# B&R Automation Studio project DevOpsDemo (part 2)

#### PackMLModuleStateManaging.cpp
```cpp
#include "PackMLModule.hpp"

		// -----------------------------------------------------------------------------

const char *internalInfoStateNames[] = { "Undefined",
	"Clearing",
	"Stopped",
	"Starting",
	"Idle",
	"Suspended",
	"Execute",
	"Stopping",
	"Aborting",
	"Aborted",
	"Holding",
	"Held",
	"Unholding",
	"Suspending",
	"Unsuspending",
	"Resetting",
	"Completing",
	"Completed",
	"",
	"",
	"",
	"",
	"",
	"",
	"",
	"",
	"",
	"",
	"",
	"",
	"Deactivating",
	"Deactivated",
	"Activating" };

const char *internalInfoModeNames[] = { "Undefined",
	"Production",
	"Maintenance",
	"Manual",
	""};

		// -----------------------------------------------------------------------------
		// we need to add complete cmd to the pattern
const unsigned long CMD_VALID_BIT_PATTERN_LIST[]
	= { 0,          0x00000080, 0x20004080, 0x000000C0, 0x000000C4, 0x0000A2C0,
	0x000092C0, 0x00000080, 0,          0x20000001, 0x000000C0, 0x000088C0,
	0x000000C0, 0x000000C0, 0x000000C0, 0x000000C0, 0x000000C0, 0x000040C0,
	0,          0,          0,          0,          0,          0,
	0,          0,          0,          0,          0,          0,
	0,          0x80000000, 0 };

// -----------------------------------------------------------------------------

PackMLModule* PackMLModule::getParentPtr(){
	if (!hasParent_)
		return nullptr;

	return pParentLink_;
}
// -----------------------------------------------------------------------------
PackMLModule* PackMLModule::getChildPtr(unsigned long int childIdx){
	if(childCount_ <= 0)
		return nullptr;

	return childLinks_[childIdx % childCount_];
}
// -----------------------------------------------------------------------------
PackMLModule* PackMLModule::getSiblingPtr(unsigned long int siblingIdx){
	if (!hasParent_)
		return nullptr;

	return pParentLink_->getChildPtr(siblingIdx);
}
// -----------------------------------------------------------------------------

PackMLModuleStateEnu PackMLModule::getChildCurrentState(unsigned long int childIndex){
	if(childCount_ <= 0)
		return ST_UNDEFINED;

	return childLinks_[childIndex % childCount_]->getCurrentState();
}
		// -----------------------------------------------------------------------------
long int PackMLModule::getChildCurrentSubState(unsigned long int childIndex){
	if(childCount_ <= 0)
		return 0;

	return childLinks_[childIndex % childCount_]->getCurrentSubState();
}
		// -----------------------------------------------------------------------------
bool PackMLModule::getChildStateComplete(unsigned long int childIndex){
	if(childCount_ <= 0)
		return false;

	return childLinks_[childIndex % childCount_]->getStateComplete();
}
		// -----------------------------------------------------------------------------
const char* PackMLModule::getChildName(unsigned long int childIndex){
	if(childCount_ <= 0)
		return "";

	return childLinks_[childIndex % childCount_]->getModuleName();
}
		// -----------------------------------------------------------------------------
PackMLModuleStateEnu PackMLModule::getSiblingCurrentState(unsigned long int siblingIndex){
	if (!hasParent_)
		return ST_UNDEFINED;

	return pParentLink_->getChildCurrentState(siblingIndex);
}
		// -----------------------------------------------------------------------------
long int PackMLModule::getSiblingCurrentSubState(unsigned long int siblingIndex){
	if (!hasParent_)
		return 0;

	return pParentLink_->getChildCurrentSubState(siblingIndex);
}
		// -----------------------------------------------------------------------------
bool PackMLModule::getSiblingStateComplete(unsigned long int siblingIndex){
	if (!hasParent_)
		return false;

	return pParentLink_->getChildStateComplete(siblingIndex);
}
		// -----------------------------------------------------------------------------
const char* PackMLModule::getSiblingName(unsigned long int siblingIndex){
	if (!hasParent_)
		return "";

	return pParentLink_->getChildName(siblingIndex);
}
		// -----------------------------------------------------------------------------
bool PackMLModule::isChild_(PackMLModule* pModule){
	for (unsigned short i = 0; i < childCount_; ++i) {
		if (childLinks_[i] == pModule) {
			return true;
		}
	}
	return false;
}
		// -----------------------------------------------------------------------------
unsigned long PackMLModule::getSiblingCount(){
	if (!hasParent_) {
		return 1;
	}
	return pParentLink_->getChildCount();
}
		// -----------------------------------------------------------------------------
bool PackMLModule::getSiblingsStateComplete(){
	if (!hasParent_) {
		return stateComplete_;
	}
	return pParentLink_->getChildrenStateComplete();
}

		// -----------------------------------------------------------------------------
bool PackMLModule::getChildrenStateComplete(){
	for (unsigned short i = 0; i < childCount_; ++i) {
		if (!childLinks_[i]->getStateComplete()) {
			return false;
		}
	}
	return true;
}
		// -----------------------------------------------------------------------------
PackMLModuleStateEnu PackMLModule::getParentCurrentState()
{
	if (!hasParent_) {
		return ST_UNDEFINED;
	}
	return pParentLink_->getCurrentState();
}

		// -----------------------------------------------------------------------------

long int PackMLModule::getParentCurrentSubState()
{
	if (!hasParent_) {
		return 0;
	}
	return pParentLink_->getCurrentSubState();
}

		// -----------------------------------------------------------------------------

const char *PackMLModule::getParentName()
{
	if (!hasParent_) {
		return "";
	}
	return pParentLink_->getModuleName();
}

bool PackMLModule::getParentStateComplete()
{
	if (!hasParent_) {
		return true;
	}
	return pParentLink_->getStateComplete();
}

		// -----------------------------------------------------------------------------

const char *PackMLModule::getCurrentStateStr() const
{
	return internalInfoStateNames[stateCurrent_];

}

const char *PackMLModule::getStateStr(PackMLModuleStateEnu state) const
{
	return internalInfoStateNames[state];
}

		// -----------------------------------------------------------------------------

		// -----------------------------------------------------------------------------

const char* PackMLModule::getCurrentModeName() const
{
	return internalInfoModeNames[modeCurrent_];
}

const char* PackMLModule::getModeName(signed long int modeId) const
{
	return internalInfoModeNames[modeId];
}

		// -----------------------------------------------------------------------------

// --------------------------------------------------------------------------

void PackMLModule::setNewModeCurrent(long int mode)
{
	modeCurrent_ = mode;

	for (unsigned short i = 0; i < childCount_; ++i) {
		childLinks_[i]->setNewModeCurrent(modeCurrent_);
	}
}

		// -----------------------------------------------------------------------------

bool PackMLModule::setCurrentMode(long int mode)
{

	// Check if the hierarchy is in synch
	if(!isModeChangePossible())
		return false;

	// update mode
	setNewModeCurrent(mode);
	// propagate mode to the children within one cycle
	return true;
}

		// -----------------------------------------------------------------------------

bool PackMLModule::isModeChangePossible()
{
	// What should the child do when it is not synchronized with the parent?
	if (!childrenInState_(stateCurrent_)) {
		return false;
	}

	for (unsigned short i = 0; i < childCount_; ++i) {
		if (!childLinks_[i]->isModeChangePossible()) {
			return false;
		}
	}

	return true;
}
		// -----------------------------------------------------------------------------

bool PackMLModule::childrenInState_(PackMLModuleStateEnu state)
{

	for (unsigned short i = 0; i < childCount_; ++i) {
		PackMLModuleStateEnu childState = childLinks_[i]->getCurrentState();
		if (childState != state && childState != ST_DEACTIVATED) {
			return false;
		}
	}
	return true;
}

		// -------------------------------------------------------------------------

bool PackMLModule::stateExistInPattern_(unsigned long stateBitPattern,
	PackMLModuleStateEnu state)
{
	if (state == ST_UNDEFINED) {
		return true;
	}
	unsigned long patternChecker = 1;
	return (stateBitPattern & (patternChecker << (state - 1)));
}

		// -------------------------------------------------------------------------

bool PackMLModule::cmdValid_(PackMLModuleStateEnu state)
{

	return stateExistInPattern_(CMD_VALID_BIT_PATTERN_LIST[stateCurrent_],
		state);
}

		// ------------------------------------------------------------------------

bool PackMLModule::isActingState(PackMLModuleStateEnu state)
{
	unsigned long actingStateBitPattern = 0xA000FAC5;

	return stateExistInPattern_(actingStateBitPattern, state);
}

		// -----------------------------------------------------------------------------

// from waiting state to acting state
void PackMLModule::executeCmd_(PackMLModuleStateEnu targetState)
{
	stateCurrent_ = targetState;
	// reset internal bools
	resetInternalCmds_();
	resetWaitingFor_();
	resetInterruptedBy_();
}

		// -----------------------------------------------------------------------------
// from acting state to waiting state
void PackMLModule::executeActingState_(PackMLModuleStateEnu targetState)
{
	if (childrenInSynch_(targetState)) {
		// Update the state
		stateCurrent_ = targetState;
		// reset internal bools
		resetInternalCmds_();
		resetWaitingFor_();
	}
}

		// -----------------------------------------------------------------------------
		// Checks if the children are in the desired state in case where they want to be
		// synchronized
bool PackMLModule::childrenInSynch_(PackMLModuleStateEnu targetState)
{

	for (unsigned long i = 0; i < childCount_; ++i) {
		if ((childLinks_[i]->getCurrentState() != targetState) && childLinks_[i]->needParentSynch(stateCurrent_)) {
			return false;
		}
	}
	return true;
}

		// -----------------------------------------------------------------------------

void PackMLModule::resetInternalCmds_()
{
	if(isActingState(stateCurrent_)){
		externalAbort_ = false;
		externalClear_ = false;
		externalStop_ = false;
		externalReset_ = false;
		externalStart_ = false;
		externalHold_ = false;
		externalUnhold_ = false;
		externalSuspend_ = false;
		externalUnsuspend_ = false;
		externalComplete_ = false;
		externalStateComplete_ = false;
	}

	activate_ = false;
	deactivate_ = false;

	abort_ = externalAbort_;
	clear_ = externalClear_;
	stop_ = externalStop_;
	reset_ = externalReset_;
	start_ = externalStart_;
	hold_ = externalHold_;
	unhold_ = externalUnhold_;
	suspend_ = externalSuspend_;
	unsuspend_ = externalUnsuspend_;
	complete_ = externalComplete_;
	stateComplete_ = false;

	oldAbort_ = false;
	oldClear_ = false;
	oldStop_ = false;
	oldReset_ = false;
	oldStart_ = false;
	oldHold_ = false;
	oldUnhold_ = false;
	oldSuspend_ = false;
	oldUnsuspend_ = false;
	oldComplete_ = false;
	oldStateComplete_ = false;

	timeInState_ = 0.0;
}

		// -----------------------------------------------------------------------------

void PackMLModule::escalateCmdAbort()
{
	if (escalateAbort_) {
		return pParentLink_->escalateCmdAbort();
	}
	abort_ = !overrideAbort_;
	externalAbort_ = abort_;
}
void PackMLModule::escalateCmdClear()
{
	if (escalateClear_) {
		return pParentLink_->escalateCmdClear();
	}
	clear_ = !overrideClear_;
	externalClear_ = clear_;
}
void PackMLModule::escalateCmdStop()
{
	if (escalateStop_) {
		return pParentLink_->escalateCmdStop();
	}
	stop_ = !overrideStop_;
	externalStop_ = stop_;
}
void PackMLModule::escalateCmdReset()
{
	if (escalateReset_) {
		return pParentLink_->escalateCmdReset();
	}
	reset_ = !overrideReset_;
	externalReset_ = reset_;
}
void PackMLModule::escalateCmdHold()
{
	if (escalateHold_) {
		return pParentLink_->escalateCmdHold();
	}
	hold_ = !overrideHold_;
	externalHold_ = hold_;
}
void PackMLModule::escalateCmdUnhold()
{
	if (escalateUnhold_) {
		return pParentLink_->escalateCmdUnhold();
	}
	unhold_ = !overrideUnhold_;
	externalUnhold_ = unhold_;
}
void PackMLModule::escalateCmdSuspend()
{
	if (escalateSuspend_) {
		return pParentLink_->escalateCmdSuspend();
	}
	suspend_ = !overrideSuspend_;
	externalSuspend_ = suspend_;
}
void PackMLModule::escalateCmdUnsuspend()
{
	if (escalateUnsuspend_) {
		return pParentLink_->escalateCmdUnsuspend();
	}
	unsuspend_ = !overrideUnsuspend_;
	externalUnsuspend_ = unsuspend_;
}
void PackMLModule::escalateCmdStart()
{
	if (escalateStart_) {
		return pParentLink_->escalateCmdStart();
	}
	start_ = !overrideStart_;
	externalStart_ = start_;
}
void PackMLModule::escalateCmdComplete()
{
	if (escalateComplete_) {
		return pParentLink_->escalateCmdComplete();
	}
	complete_ = !overrideComplete_;
	externalComplete_ = complete_;
}

// ----------------------------------------------------------------------------

void PackMLModule::propagateCmdAbort(bool root)
{
	abort_ = reactToAbort_ && !root;
	externalAbort_ = abort_;

	for (unsigned short i = 0; i < childCount_; ++i) {
		childLinks_[i]->propagateCmdAbort(false);
	}
}
void PackMLModule::propagateCmdClear(bool root)
{
	clear_ = reactToClear_ && !root;
	externalClear_ = clear_;

	for (unsigned short i = 0; i < childCount_; ++i) {
		childLinks_[i]->propagateCmdClear(false);
	}
}
void PackMLModule::propagateCmdStop(bool root)
{
	stop_ = reactToStop_ && !root;
	externalStop_ = stop_;

	for (unsigned short i = 0; i < childCount_; ++i) {
		childLinks_[i]->propagateCmdStop(false);
	}
}
void PackMLModule::propagateCmdReset(bool root)
{
	reset_ = reactToReset_ && !root;
	externalReset_ = reset_;

	for (unsigned short i = 0; i < childCount_; ++i) {
		childLinks_[i]->propagateCmdReset(false);
	}
}
void PackMLModule::propagateCmdHold(bool root)
{
	hold_ = reactToHold_ && !root;
	externalHold_ = hold_;

	for (unsigned short i = 0; i < childCount_; ++i) {
		childLinks_[i]->propagateCmdHold(false);
	}
}
void PackMLModule::propagateCmdUnhold(bool root)
{
	unhold_ = reactToUnhold_ && !root;
	externalUnhold_ = unhold_;

	for (unsigned short i = 0; i < childCount_; ++i) {
		childLinks_[i]->propagateCmdUnhold(false);
	}
}
void PackMLModule::propagateCmdSuspend(bool root)
{
	suspend_ = reactToSuspend_ && !root;
	externalSuspend_ = suspend_;

	for (unsigned short i = 0; i < childCount_; ++i) {
		childLinks_[i]->propagateCmdSuspend(false);
	}
}
void PackMLModule::propagateCmdUnsuspend(bool root)
{
	unsuspend_ = reactToUnsuspend_ && !root;
	externalUnsuspend_ = unsuspend_;

	for (unsigned short i = 0; i < childCount_; ++i) {
		childLinks_[i]->propagateCmdUnsuspend(false);
	}
}
void PackMLModule::propagateCmdStart(bool root)
{
	start_ = reactToStart_ && !root;
	externalStart_ = start_;

	for (unsigned short i = 0; i < childCount_; ++i) {
		childLinks_[i]->propagateCmdStart(false);
	}
}
void PackMLModule::propagateCmdComplete(bool root)
{
	complete_ = reactToComplete_ && !root;
	externalComplete_ = complete_;

	for (unsigned short i = 0; i < childCount_; ++i) {
		childLinks_[i]->propagateCmdComplete(false);
	}
}

// ----------------------------------------------------------------------------

bool PackMLModule::evaluateCmdAbort(bool& newCmd)
{
	if (newCmd && !oldAbort_) {
		oldAbort_ = true;
		return setCmd_(ST_ABORTING);
	}
	else if (!newCmd && oldAbort_) {
		oldAbort_ = false;
		resetCmd_(ST_ABORTING);
	}
	return true;
}
bool PackMLModule::evaluateCmdStop(bool& newCmd)
{
	if (newCmd && !oldStop_) {
		oldStop_ = true;
		return setCmd_(ST_STOPPING);
	}
	else if (!newCmd && oldStop_) {
		oldStop_ = false;
		resetCmd_(ST_STOPPING);
	}
	return true;
}
bool PackMLModule::evaluateCmdClear(bool& newCmd)
{
	if (newCmd && !oldClear_) {
		oldClear_ = true;
		return setCmd_(ST_CLEARING);
	}
	else if (!newCmd && oldClear_) {
		oldClear_ = false;
		resetCmd_(ST_CLEARING);
	}
	return true;
}
bool PackMLModule::evaluateCmdReset(bool& newCmd)
{
	if (newCmd && !oldReset_) {
		oldReset_ = true;
		return setCmd_(ST_RESETTING);
	}
	else if (!newCmd && oldReset_) {
		oldReset_ = false;
		resetCmd_(ST_RESETTING);
	}
	return true;
}
bool PackMLModule::evaluateCmdStart(bool& newCmd)
{
	if (newCmd && !oldStart_) {
		oldStart_ = true;
		return setCmd_(ST_STARTING);
	}
	else if (!newCmd && oldStart_) {
		oldStart_ = false;
		resetCmd_(ST_STARTING);
	}
	return true;
}
bool PackMLModule::evaluateCmdSuspend(bool& newCmd)
{
	if (newCmd && !oldSuspend_) {
		oldSuspend_ = true;
		return setCmd_(ST_SUSPENDING);
	}
	else if (!newCmd && oldSuspend_) {
		oldSuspend_ = false;
		resetCmd_(ST_SUSPENDING);
	}
	return true;
}
bool PackMLModule::evaluateCmdUnsuspend(bool& newCmd)
{
	if (newCmd && !oldUnsuspend_) {
		oldUnsuspend_ = true;
		return setCmd_(ST_UNSUSPENDING);
	}
	else if (!newCmd && oldUnsuspend_) {
		oldUnsuspend_ = false;
		resetCmd_(ST_UNSUSPENDING);
	}
	return true;
}
bool PackMLModule::evaluateCmdHold(bool& newCmd)
{
	if (newCmd && !oldHold_) {
		oldHold_ = true;
		return setCmd_(ST_HOLDING);
	}
	else if (!newCmd && oldHold_) {
		oldHold_ = false;
		resetCmd_(ST_HOLDING);
	}
	return true;
}
bool PackMLModule::evaluateCmdUnhold(bool& newCmd)
{
	if (newCmd && !oldUnhold_) {
		oldUnhold_ = true;
		return setCmd_(ST_UNHOLDING);
	}
	else if (!newCmd && oldUnhold_) {
		oldUnhold_ = false;
		resetCmd_(ST_UNHOLDING);
	}
	return true;
}
bool PackMLModule::evaluateCmdComplete(bool& newCmd)
{
	if (newCmd && !oldComplete_) {
		oldComplete_ = true;
		return setCmd_(ST_COMPLETING);
	}
	else if (!newCmd && oldComplete_) {
		oldComplete_ = false;
		resetCmd_(ST_COMPLETING);
	}
	return true;
}
bool PackMLModule::evaluateCmdStateComplete(bool& newCmd)
{
	if (newCmd && !oldStateComplete_) {
		oldStateComplete_ = true;
		return setCmd_(ST_UNDEFINED);
	}
	else if (!newCmd && oldStateComplete_) {
		oldStateComplete_ = false;
		resetCmd_(ST_UNDEFINED);
	}
	return true;
}

bool PackMLModule::setCmdAbort(){
	return setCmd_(ST_ABORTING);
}
bool PackMLModule::setCmdStop(){
	return setCmd_(ST_STOPPING);
}
bool PackMLModule::setCmdClear(){
	return setCmd_(ST_CLEARING);
}
bool PackMLModule::setCmdReset(){
	return setCmd_(ST_RESETTING);
}
bool PackMLModule::setCmdStart(){
	return setCmd_(ST_STARTING);
}
bool PackMLModule::setCmdSuspend(){
	return setCmd_(ST_SUSPENDING);
}
bool PackMLModule::setCmdUnsuspend(){
	return setCmd_(ST_UNSUSPENDING);
}
bool PackMLModule::setCmdHold(){
	return setCmd_(ST_HOLDING);
}
bool PackMLModule::setCmdUnhold(){
	return setCmd_(ST_UNHOLDING);
}
bool PackMLModule::setCmdComplete(){
	return setCmd_(ST_COMPLETING);
}
bool PackMLModule::setCmdStateComplete(){
	return setCmd_(ST_UNDEFINED);
}

void PackMLModule::resetCmdAbort(){
	return resetCmd_(ST_ABORTING);
}
void PackMLModule::resetCmdStop(){
	return resetCmd_(ST_STOPPING);
}
void PackMLModule::resetCmdClear(){
	return resetCmd_(ST_CLEARING);
}
void PackMLModule::resetCmdReset(){
	return resetCmd_(ST_RESETTING);
}
void PackMLModule::resetCmdStart(){
	return resetCmd_(ST_STARTING);
}
void PackMLModule::resetCmdSuspend(){
	return resetCmd_(ST_SUSPENDING);
}
void PackMLModule::resetCmdUnsuspend(){
	return resetCmd_(ST_UNSUSPENDING);
}
void PackMLModule::resetCmdHold(){
	return resetCmd_(ST_HOLDING);
}
void PackMLModule::resetCmdUnhold(){
	return resetCmd_(ST_UNHOLDING);
}
void PackMLModule::resetCmdComplete(){
	return resetCmd_(ST_COMPLETING);
}
void PackMLModule::resetCmdStateComplete(){
	return resetCmd_(ST_UNDEFINED);
}

		// -----------------------------------------------------------------------------

bool PackMLModule::setCmd_(PackMLModuleStateEnu targetActingState) // NOLINT
{

	bool cmdValid = cmdValid_(targetActingState);

	switch (targetActingState) { // NOCCM
		case ST_CLEARING:
			if (overrideClear_ && !escalateClear_) {
				return false; // error code
			}
			if (hasParent_ && escalateClear_ && cmdValid) {
				pParentLink_->escalateCmdClear();
				setInterruptedBy_(ST_CLEARING);
			}
			clear_ = !overrideClear_; //!overrideAbort_ || !escalateAbort_;
			break;

		case ST_STARTING:
			if (overrideStart_ && !escalateStart_) {
				return false; // error code
			}
			if (hasParent_ && escalateStart_ && cmdValid) {
				pParentLink_->escalateCmdStart();
				setInterruptedBy_(ST_STARTING);
			}
			start_ = !overrideStart_;
			break;

		case ST_STOPPING:
			if (overrideStop_ && !escalateStop_) {
				return false; // error code
			}
			if (hasParent_ && escalateStop_) {
				pParentLink_->escalateCmdStop();
			}
			if(cmdValid){
				setInterruptedBy_(ST_STOPPING);
				stop_ = !overrideStop_;
			}
			break;

		case ST_ABORTING:
			if (overrideAbort_ && !escalateAbort_) {
				return false; // error code
			}
			if (hasParent_ && escalateAbort_) {
				pParentLink_->escalateCmdAbort();
			}

			if(cmdValid){
				setInterruptedBy_(ST_ABORTING);
				abort_ = !overrideAbort_;
			}
			break;

		case ST_HOLDING:
			if (overrideHold_ && !escalateHold_) {
				return false; // error code
			}
			if (hasParent_ && escalateHold_) {
				pParentLink_->escalateCmdHold();
			}
			if(cmdValid){
				setInterruptedBy_(ST_HOLDING);
				hold_ = !overrideHold_;
			}
			break;

		case ST_UNHOLDING:
			if (overrideUnhold_ && !escalateUnhold_) {
				return false; // error code
			}
			if (hasParent_ && escalateUnhold_ && cmdValid) {
				pParentLink_->escalateCmdUnhold();
				setInterruptedBy_(ST_UNHOLDING);
			}
			unhold_ = !overrideUnhold_;
			break;

		case ST_SUSPENDING:
			if (overrideSuspend_ && !escalateSuspend_) {
				return false; // error code
			}
			if (hasParent_ && escalateSuspend_) {
				pParentLink_->escalateCmdSuspend();
			}
			if(cmdValid){
				setInterruptedBy_(ST_SUSPENDING);
				suspend_ = !overrideSuspend_;
			}
			break;

		case ST_UNSUSPENDING:
			if (overrideUnsuspend_ && !escalateUnsuspend_) {
				return false; // error code
			}
			if (hasParent_ && escalateUnsuspend_ && cmdValid) {
				pParentLink_->escalateCmdUnsuspend();
				setInterruptedBy_(ST_UNSUSPENDING);
			}
			unsuspend_ = !overrideUnsuspend_;
			break;

		case ST_RESETTING:
			if (overrideReset_ && !escalateReset_) {
				return false; // error code
			}
			if (hasParent_ && escalateReset_ && cmdValid) {
				pParentLink_->escalateCmdReset();
				setInterruptedBy_(ST_RESETTING);
			}
			reset_ = !overrideReset_;
			break;

		case ST_COMPLETING:
			// check if the state group is configured
			if (overrideComplete_ && !escalateComplete_) {
				return false; // error code
			}
			if (hasParent_ && escalateComplete_) {
				pParentLink_->escalateCmdComplete();
			}
			if(cmdValid){
				setInterruptedBy_(ST_COMPLETING);
				complete_ = !overrideComplete_;
			}
			break;

		case ST_UNDEFINED:
			stateComplete_ = true;
			break;

		default:
			break;
	}

	return true;
}

		// -----------------------------------------------------------------------------

void PackMLModule::resetCmd_(PackMLModuleStateEnu targetActingState)
{

	switch (targetActingState) { // NOCCM
		case ST_CLEARING:
			clear_ = externalClear_;
			break;

		case ST_STARTING:
			start_ = externalStart_;
			break;

		case ST_STOPPING:
			stop_ = externalStop_;
			break;

		case ST_ABORTING:
			abort_ = externalAbort_;
			break;

		case ST_HOLDING:
			hold_ = externalHold_;
			break;

		case ST_UNHOLDING:
			unhold_ = externalUnhold_;
			break;

		case ST_SUSPENDING:
			suspend_ = externalSuspend_;
			break;

		case ST_UNSUSPENDING:
			unsuspend_ = externalUnsuspend_;
			break;

		case ST_RESETTING:
			reset_ = externalReset_;
			break;

		case ST_COMPLETING:
			complete_ = externalComplete_;
			break;

		case ST_UNDEFINED:
			stateComplete_ = externalStateComplete_;
			break;

		default:
			break;
	}
}

		// -----------------------------------------------------------------------------

		// if parent synchronization needed
bool PackMLModule::needParentSynch(PackMLModuleStateEnu state)
{
	if (hierarchyLevel_ == 0) {
		return true;
	}

	switch (stateCurrent_) { // NOCCM

		case ST_CLEARING:
			switch (state) { // NOCCM
				case ST_ABORTING:
					return overrideAbort_ || reactToAbort_;
				case ST_CLEARING:
					return overrideClear_ || reactToClear_;
				default:
					break;
			}
			break;

		case ST_STOPPED:
			switch (state) { // NOCCM
				case ST_ABORTING:
					return overrideAbort_ || reactToAbort_;
				case ST_RESETTING:
					return overrideReset_ || reactToReset_;
				default:
					break;
			}
			break;

		case ST_IDLE:
			switch (state) { // NOCCM
				case ST_ABORTING:
					return overrideAbort_ || reactToAbort_;
				case ST_STOPPING:
					return overrideStop_ || reactToStop_;
				case ST_STARTING:
					return overrideStart_ || reactToStart_;
				default:
					break;
			}
			break;

		case ST_SUSPENDED:
			switch (state) { // NOCCM
				case ST_ABORTING:
					return overrideAbort_ || reactToAbort_;
				case ST_STOPPING:
					return overrideStop_ || reactToStop_;
				case ST_UNSUSPENDING:
					return overrideUnsuspend_ || reactToUnsuspend_;
				case ST_HOLDING:
					return overrideHold_ || reactToHold_;
				case ST_COMPLETING:
					return overrideComplete_ || reactToComplete_;
				default:
					break;
			}
			break;

		case ST_EXECUTE:
			switch (state) { // NOCCM
				case ST_ABORTING:
					return overrideAbort_ || reactToAbort_;
				case ST_STOPPING:
					return overrideStop_ || reactToStop_;
				case ST_SUSPENDING:
					return overrideSuspend_ || reactToSuspend_;
				case ST_HOLDING:
					return overrideHold_ || reactToHold_;
				case ST_COMPLETING:
					return overrideComplete_ || reactToComplete_;
				default:
					break;
			}
			break;

		case ST_STOPPING:
			switch (state) { // NOCCM
				case ST_ABORTING:
					return overrideAbort_ || reactToAbort_;
				case ST_STOPPING:
					return overrideStop_ || reactToStop_;
				default:
					break;
			}
			break;

		case ST_ABORTING:
			switch (state) { // NOCCM
				case ST_ABORTING:
					return overrideAbort_ || reactToAbort_;
				default:
					break;
			}
			break;

		case ST_ABORTED:
			switch (state) { // NOCCM
				case ST_CLEARING:
					return overrideClear_ || reactToClear_;
				default:
					break;
			}
			break;

		case ST_HELD:
			switch (state) { // NOCCM
				case ST_ABORTING:
					return overrideAbort_ || reactToAbort_;
				case ST_STOPPING:
					return overrideStop_ || reactToStop_;
				case ST_UNHOLDING:
					return overrideUnhold_ || reactToUnhold_;
				case ST_COMPLETING:
					return overrideComplete_ || reactToComplete_;
				default:
					break;
			}
			break;

		case ST_SUSPENDING:
			switch (state) { // NOCCM
				case ST_ABORTING:
					return overrideAbort_ || reactToAbort_;
				case ST_STOPPING:
					return overrideStop_ || reactToStop_;
				case ST_SUSPENDING:
					return overrideSuspend_ || reactToSuspend_;
				default:
					break;
			}
			break;
		case ST_UNSUSPENDING:
			switch (state) { // NOCCM
				case ST_ABORTING:
					return overrideAbort_ || reactToAbort_;
				case ST_STOPPING:
					return overrideStop_ || reactToStop_;
				case ST_UNSUSPENDING:
					return overrideUnsuspend_ || reactToUnsuspend_;
				default:
					break;
			}
			break;
		case ST_COMPLETING:
			switch (state) { // NOCCM
				case ST_ABORTING:
					return overrideAbort_ || reactToAbort_;
				case ST_STOPPING:
					return overrideStop_ || reactToStop_;
				case ST_COMPLETING:
					return overrideComplete_ || reactToComplete_;
				default:
					break;
			}
			break;
		case ST_STARTING:
			switch (state) { // NOCCM
				case ST_ABORTING:
					return overrideAbort_ || reactToAbort_;
				case ST_STOPPING:
					return overrideStop_ || reactToStop_;
				case ST_STARTING:
					return overrideStart_ || reactToStart_;
				default:
					break;
			}
			break;
		case ST_HOLDING:
			switch (state) { // NOCCM
				case ST_ABORTING:
					return overrideAbort_ || reactToAbort_;
				case ST_STOPPING:
					return overrideStop_ || reactToStop_;
				case ST_HOLDING:
					return overrideHold_ || reactToHold_;
				default:
					break;
			}
			break;
		case ST_UNHOLDING:
			switch (state) { // NOCCM
				case ST_ABORTING:
					return overrideAbort_ || reactToAbort_;
				case ST_STOPPING:
					return overrideStop_ || reactToStop_;
				case ST_UNHOLDING:
					return overrideUnhold_ || reactToUnhold_;
				default:
					break;
			}
			break;

		case ST_RESETTING:
			switch (state) { // NOCCM
				case ST_ABORTING:
					return overrideAbort_ || reactToAbort_;
				case ST_STOPPING:
					return overrideStop_ || reactToStop_;
				case ST_RESETTING:
					return overrideReset_ || reactToReset_;
				default:
					break;
			}
			break;

		case ST_COMPLETE:
			switch (state) { // NOCCM
				case ST_ABORTING:
					return overrideAbort_ || reactToAbort_;
				case ST_STOPPING:
					return overrideStop_ || reactToStop_;
				case ST_RESETTING:
					return overrideReset_ || reactToReset_;
				default:
					break;
			}
			break;

		default:
			break;
	}

	return false;
}

// -----------------------------------------------------------------------------
// decide if reacto to only should when parent + 1 state in front of child. e.g. instead of ST_ABORTING and ST_ABORTED --> only ST_ABORTING
void PackMLModule::checkParentStateCondition_()
{
	if (hierarchyLevel_ == 0) {
		return;
	}

	PackMLModuleStateEnu parentState = getParentCurrentState();

	if (parentState == stateCurrent_) {
		return;
	}

	switch (stateCurrent_) { // NOCCM
		case ST_CLEARING:
			switch (parentState) { // NOCCM
				case ST_ABORTING:
					abort_ = overrideAbort_ || abort_ || reactToAbort_;
					break;
				case ST_ABORTED:
					abort_ = overrideAbort_ || abort_;
					break;
				default:
					break;
			}
			break;

		case ST_STOPPED:
			switch (parentState) { // NOCCM
				case ST_ABORTING:
					abort_ = overrideAbort_ || abort_ || reactToAbort_;
					break;
				case ST_ABORTED:
					abort_ = overrideAbort_ || abort_;
					break;

				case ST_DEACTIVATING:
				case ST_DEACTIVATED:
					deactivate_ = (activationCondition_ == 1);
					break;

				case ST_RESETTING:
					reset_ = overrideReset_ || reset_ || reactToReset_;
					break;

				case ST_IDLE:
				case ST_STARTING:
				case ST_SUSPENDED:
				case ST_EXECUTE:
				case ST_HOLDING:
				case ST_HELD:
				case ST_UNHOLDING:
				case ST_SUSPENDING:
				case ST_UNSUSPENDING:
				case ST_COMPLETING:
				case ST_COMPLETE:
					reset_ = overrideReset_ || reset_;
					break;

				default:
					break;
			}
			break;

		case ST_IDLE:
			switch (parentState) { // NOCCM
				case ST_ABORTING:
					abort_ = overrideAbort_ || abort_ || reactToAbort_;
					break;
				case ST_ABORTED:
					abort_ = overrideAbort_ || abort_;
					break;

				case ST_CLEARING:
					stop_ = overrideStop_ || stop_;
					abort_ = (overrideAbort_ || abort_) && !stop_;
					break;

				case ST_STOPPING:
					stop_ = overrideStop_ || stop_ || reactToStop_;
					break;
				case ST_STOPPED:
					stop_ = overrideStop_ || stop_;
					break;

				case ST_DEACTIVATING:
				case ST_DEACTIVATED:
				case ST_ACTIVATING:
					stop_ = overrideStop_ || stop_;
					abort_ = (overrideAbort_ || abort_) && !stop_;
					break;

				case ST_STARTING:
					start_ = overrideStart_ || start_ || reactToStart_;
					break;

				case ST_EXECUTE:
				case ST_SUSPENDED:
				case ST_HOLDING:
				case ST_HELD:
				case ST_UNHOLDING:
				case ST_SUSPENDING:
				case ST_UNSUSPENDING:
				case ST_COMPLETING:
				case ST_COMPLETE:
					start_ = overrideStart_ || start_;
					break;

				default:
					break;
			}
			break;

		case ST_SUSPENDED:
			switch (parentState) { // NOCCM
				case ST_ABORTING:
					abort_ = overrideAbort_ || abort_ || reactToAbort_;
					break;
				case ST_ABORTED:
					abort_ = overrideAbort_ || abort_;
					break;

				case ST_CLEARING:
					stop_ = overrideStop_ || stop_;
					abort_ = (overrideAbort_ || abort_) && !stop_;
					break;

				case ST_STOPPING:
					stop_ = overrideStop_ || stop_ || reactToStop_;
					break;
				case ST_STOPPED:
					stop_ = overrideStop_ || stop_;
					break;

				case ST_UNSUSPENDING:
					unsuspend_ = overrideUnsuspend_ || unsuspend_ || reactToUnsuspend_;
					break;

				case ST_DEACTIVATING:
				case ST_DEACTIVATED:
				case ST_ACTIVATING:
					stop_ = overrideStop_ || stop_;
					abort_ = (overrideAbort_ || abort_) && !stop_;
					break;

				case ST_RESETTING:
				case ST_IDLE: // **********************
					unsuspend_ = overrideUnsuspend_ || unsuspend_;
					stop_ = (overrideStop_ || stop_) && !unsuspend_;
					break;

				case ST_COMPLETING:
					complete_ = overrideComplete_ || complete_ || reactToComplete_;
					break;
				case ST_COMPLETE:
					complete_ = overrideComplete_ || complete_;
					break;

				case ST_HOLDING:
					hold_ = overrideHold_ || hold_ || reactToHold_;
					break;
				case ST_HELD:
					hold_ = overrideHold_ || hold_;
					break;

				case ST_EXECUTE:
				case ST_STARTING:
				case ST_UNHOLDING:
					unsuspend_ = overrideUnsuspend_ || unsuspend_;
					break;

				default:
					break;
			}
			break;

		case ST_EXECUTE:
			switch (parentState) { // NOCCM
				case ST_ABORTING:
					abort_ = overrideAbort_ || abort_ || reactToAbort_;
					break;
				case ST_ABORTED:
					abort_ = overrideAbort_ || abort_;
					break;

				case ST_CLEARING:
					stop_ = overrideStop_ || stop_;
					abort_ = (overrideAbort_ || abort_) && !stop_;
					break;

				case ST_STOPPING:
					stop_ = overrideStop_ || stop_ || reactToStop_;
					break;

				case ST_STOPPED:
					stop_ = overrideStop_ || stop_;
					break;

				case ST_SUSPENDING:
					suspend_ = overrideSuspend_ || suspend_ || reactToSuspend_;
					break;

				case ST_SUSPENDED:
					suspend_ = overrideSuspend_ || suspend_;
					break;

				case ST_HOLDING:
					hold_ = overrideHold_ || hold_ || reactToHold_;
					break;

				case ST_HELD:
					hold_ = overrideHold_ || hold_;
					break;

				case ST_COMPLETING:
					complete_ = overrideComplete_ || complete_ || reactToComplete_;
					break;

				case ST_COMPLETE:
					complete_ = overrideComplete_ || complete_;
					break;

				case ST_DEACTIVATING:
				case ST_DEACTIVATED:
				case ST_ACTIVATING:
					stop_ = overrideStop_ || stop_;
					abort_ = (overrideAbort_ || abort_) && !stop_;
					break;

				case ST_RESETTING:
				case ST_IDLE:
					complete_ = overrideComplete_ || complete_;
					stop_ = (overrideStop_ || stop_) && !complete_;
					break;

				default:
					break;
			}
			break;

		case ST_STOPPING:
			switch (parentState) { // NOCCM
				case ST_ABORTING:
					abort_ = overrideAbort_ || abort_ || reactToAbort_;
					break;
				case ST_ABORTED:
					abort_ = overrideAbort_ || abort_;
					break;
				default:
					break;
			}
			break;

		case ST_ABORTED:
			switch (parentState) { // NOCCM
				case ST_DEACTIVATING:
				case ST_DEACTIVATED:
					deactivate_ = (activationCondition_ == 1);
					break;

				case ST_CLEARING:
					clear_ = overrideClear_ || clear_ || reactToClear_;
					break;

				case ST_STOPPED:
				case ST_STARTING:
				case ST_IDLE:
				case ST_SUSPENDED:
				case ST_EXECUTE:
				case ST_STOPPING:
				case ST_HOLDING:
				case ST_HELD:
				case ST_UNHOLDING:
				case ST_SUSPENDING:
				case ST_UNSUSPENDING:
				case ST_RESETTING:
				case ST_COMPLETING:
				case ST_COMPLETE:
				case ST_ACTIVATING:
					clear_ = overrideClear_ || clear_;
					break;

				default:
					break;
			}
			break;

		case ST_HELD:
			switch (parentState) { // NOCCM
				case ST_ABORTING:
					abort_ = overrideAbort_ || abort_ || reactToAbort_;
					break;
				case ST_ABORTED:
					abort_ = overrideAbort_ || abort_;
					break;

				case ST_CLEARING:
					stop_ = overrideStop_ || stop_;
					abort_ = (overrideAbort_ || abort_) && !stop_;
					break;

				case ST_STOPPING:
					stop_ = overrideStop_ || stop_ || reactToStop_;
					break;

				case ST_STOPPED:
					stop_ = overrideStop_ || stop_;
					break;

				case ST_UNHOLDING:
					unhold_ = overrideUnhold_ || unhold_ || reactToUnhold_;
					break;

				case ST_DEACTIVATING:
				case ST_DEACTIVATED:
				case ST_ACTIVATING:
					stop_ = overrideStop_ || stop_;
					abort_ = (overrideAbort_ || abort_) && !stop_;
					break;

				case ST_RESETTING:
				case ST_IDLE: // **********************
					unhold_ = overrideUnhold_ || unhold_;
					stop_ = (overrideStop_ || stop_) && !unhold_;
					break;

				case ST_COMPLETING:
					complete_ = overrideComplete_ || complete_ || reactToComplete_;
					break;
				case ST_COMPLETE:
					complete_ = overrideComplete_ || complete_;
					break;

				case ST_EXECUTE:
				case ST_SUSPENDING:
				case ST_SUSPENDED:
				case ST_UNSUSPENDING:
				case ST_STARTING:
					unhold_ = overrideUnhold_ || unhold_;
					break;

				default:
					break;
			}
			break;

		case ST_STARTING:
		case ST_HOLDING:
		case ST_UNHOLDING:
		case ST_SUSPENDING:
		case ST_UNSUSPENDING:
			switch (parentState) { // NOCCM
				case ST_ABORTING:
					abort_ = overrideAbort_ || abort_ || reactToAbort_;
					break;

				case ST_ABORTED:
					abort_ = overrideAbort_ || abort_;
					break;

				case ST_CLEARING:
					stop_ = overrideStop_ || stop_;
					abort_ = (overrideAbort_ || abort_) && !stop_;
					break;

				case ST_STOPPING:
					stop_ = overrideStop_ || stop_ || reactToStop_;
					break;

				case ST_STOPPED:
					stop_ = overrideStop_ || stop_;
					break;

				case ST_DEACTIVATING:
				case ST_DEACTIVATED:
				case ST_ACTIVATING:
					stop_ = overrideStop_ || stop_;
					abort_ = (overrideAbort_ || abort_) && !stop_;
					break;

				case ST_RESETTING:
				case ST_IDLE:
					stop_ = overrideStop_ || stop_;
					break;

				default:
					break;
			}
			break;

		case ST_RESETTING:
		case ST_COMPLETING:
			switch (parentState) { // NOCCM
				case ST_ABORTING:
					abort_ = overrideAbort_ || abort_ || reactToAbort_;
					break;
				case ST_ABORTED:
					abort_ = overrideAbort_ || abort_;
					break;

				case ST_CLEARING:
					stop_ = overrideStop_ || stop_;
					abort_ = (overrideAbort_ || abort_) && !stop_;
					break;

				case ST_STOPPING:
					stop_ = overrideStop_ || stop_ || reactToStop_;
					break;

				case ST_STOPPED:
					stop_ = overrideStop_ || stop_;
					break;

				case ST_DEACTIVATING:
				case ST_DEACTIVATED:
				case ST_ACTIVATING:
					stop_ = overrideStop_ || stop_;
					abort_ = (overrideAbort_ || abort_) && !stop_;
					break;

				default:
					break;
			}
			break;

		case ST_COMPLETE:
			switch (parentState) { // NOCCM
				case ST_ABORTING:
					abort_ = overrideAbort_ || abort_ || reactToAbort_;
					break;
				case ST_ABORTED:
					abort_ = overrideAbort_ || abort_;
					break;

				case ST_CLEARING:
					stop_ = overrideStop_ || stop_;
					abort_ = (overrideAbort_ || abort_) && !stop_;
					break;

				case ST_STOPPING:
					stop_ = overrideStop_ || stop_ || reactToStop_;
					break;

				case ST_STOPPED:
					stop_ = overrideStop_ || stop_;
					break;

				case ST_DEACTIVATING:
				case ST_DEACTIVATED:
				case ST_ACTIVATING:
					stop_ = overrideStop_ || stop_;
					abort_ = (overrideAbort_ || abort_) && !stop_;
					break;

				case ST_RESETTING:
					reset_ = overrideReset_ || reset_ || reactToReset_;
					break;

				case ST_IDLE:
				case ST_STARTING:
				case ST_SUSPENDED:
				case ST_EXECUTE:
				case ST_HOLDING:
				case ST_HELD:
				case ST_UNHOLDING:
				case ST_SUSPENDING:
				case ST_UNSUSPENDING:
					reset_ = overrideReset_ || reset_;
					break;

				default:
					break;
			}
			break;

		case ST_DEACTIVATED:
			if (parentState != ST_DEACTIVATING) {
				activate_ = (activationCondition_ == 1);
			}
			break;

		default:
			break;
	}

}

void PackMLModule::resetWaitingFor_()
{
	if((waitingForIndex_ == moduleIndex_) && hasParent_){
		pParentLink_->escalateResetWaitingFor(moduleIndex_);
	}

	waitingForIndex_ = 0xFFFFFFFF;
	waitingForLevel_ = 0;
}

void PackMLModule::escalateResetWaitingFor(unsigned long int waitingForIndex){

	if(waitingForIndex == waitingForIndex_){
		waitingForIndex_ = 0xFFFFFFFF;
		waitingForLevel_ = 0;
	}

	if(hasParent_){
		pParentLink_->escalateResetWaitingFor(waitingForIndex);
	}

}

void PackMLModule::setWaitingFor_(PackMLModuleStateEnu cmdState)
{
	// escallate
	if(hierarchyLevel_ >= waitingForLevel_){
		waitingForIndex_ = moduleIndex_;
		waitingForLevel_ = hierarchyLevel_;

		if(hasParent_ && needParentSynch(cmdState)){
			pParentLink_->escalateWaitingFor(waitingForIndex_, waitingForLevel_, cmdState);
		}
	}
}

void PackMLModule::escalateWaitingFor(unsigned long int waitingForIndex, unsigned short int waitingForLevel, PackMLModuleStateEnu cmdState){

	if(waitingForLevel >= waitingForLevel_){
		waitingForIndex_ = waitingForIndex;
		waitingForLevel_ = waitingForLevel;

		if(hasParent_ && needParentSynch(cmdState)){
			pParentLink_->escalateWaitingFor(waitingForIndex_, waitingForLevel_, cmdState);
		}
	}
}

//void PackMLModule::escalateWaitingFor(unsigned long int moduleIndex)
//{
//	if (escalateStart_) {
//		return pParentLink_->escalateCmdStart();
//	}
//}

	//	 -----------------------------------------------------------------------------

void PackMLModule::resetInterruptedBy_()
{
	switch(interruptedInState_){
		case ST_EXECUTE:
			if(stateCurrent_ == ST_ABORTING || stateCurrent_ == ST_SUSPENDING || stateCurrent_ == ST_HOLDING || stateCurrent_ == ST_STOPPING || stateCurrent_ == ST_COMPLETING)
				return;
			break;

		case ST_STOPPED:
			if(stateCurrent_ == ST_ABORTING || stateCurrent_ == ST_RESETTING)
				return;
			break;

		case ST_IDLE:
			if(stateCurrent_ == ST_ABORTING || stateCurrent_ == ST_STOPPING || stateCurrent_ == ST_STARTING)
				return;
			break;

		case ST_HELD:
			if(stateCurrent_ == ST_ABORTING || stateCurrent_ == ST_STOPPING || stateCurrent_ == ST_UNHOLDING)
				return;
			break;

		case ST_SUSPENDED:
			if(stateCurrent_ == ST_ABORTING || stateCurrent_ == ST_STOPPING || stateCurrent_ == ST_UNSUSPENDING)
				return;
			break;

		case ST_ABORTED:
			if(stateCurrent_ == ST_CLEARING)
				return;
			break;

		case ST_COMPLETE:
			if(stateCurrent_ == ST_ABORTING || stateCurrent_ == ST_STOPPING || stateCurrent_ == ST_RESETTING)
				return;
			break;

	//	case ST_RESETTING: ST_STARTING: ST_HOLDING: ST_UNHOLDING: ST_SUSPENDING: ST_UNSUSPENDING: ST_COMPLETING: ST_STOPPING: ST_ABORTING: ST_CLEARING:
		default:
			if(stateCurrent_ == ST_ABORTING || stateCurrent_ == ST_STOPPING)
				return;
			break;
	}

	interruptedByIndex_ = 0xFFFFFFFF;
	interruptedInState_ = ST_UNDEFINED;
	interruptedInSubState_ = 0;
}

void PackMLModule::setInterruptedBy_(PackMLModuleStateEnu cmdState)
{
	escalateInterruptedBy(moduleIndex_, stateCurrent_, subStateCurrent_, cmdState);
}

void PackMLModule::escalateInterruptedBy(unsigned long int moduleIndex, PackMLModuleStateEnu state, signed long int subState, PackMLModuleStateEnu cmdState)
{
	switch (cmdState) { // NOCCM
		case ST_CLEARING:
			if (hasParent_ && escalateClear_) {
				return pParentLink_->escalateInterruptedBy(moduleIndex, state, subState, cmdState);
			}
			break;

		case ST_STARTING:
			if (hasParent_ && escalateStart_) {
				return pParentLink_->escalateInterruptedBy(moduleIndex, state, subState, cmdState);
			}
			break;

		case ST_STOPPING:
			if (hasParent_ && escalateStop_) {
				return pParentLink_->escalateInterruptedBy(moduleIndex, state, subState, cmdState);
			}
			break;

		case ST_ABORTING:
			if (hasParent_ && escalateAbort_) {
				return pParentLink_->escalateInterruptedBy(moduleIndex, state, subState, cmdState);
			}
			break;

		case ST_HOLDING:
			if (hasParent_ && escalateHold_) {
				return pParentLink_->escalateInterruptedBy(moduleIndex, state, subState, cmdState);
			}
			break;

		case ST_UNHOLDING:
			if (hasParent_ && escalateUnhold_) {
				return pParentLink_->escalateInterruptedBy(moduleIndex, state, subState, cmdState);
			}
			break;

		case ST_SUSPENDING:
			if (hasParent_ && escalateSuspend_) {
				return pParentLink_->escalateInterruptedBy(moduleIndex, state, subState, cmdState);
			}
			break;

		case ST_UNSUSPENDING:
			if (hasParent_ && escalateUnsuspend_) {
				return pParentLink_->escalateInterruptedBy(moduleIndex, state, subState, cmdState);
			}
			break;

		case ST_RESETTING:
			if (hasParent_ && escalateReset_) {
				return pParentLink_->escalateInterruptedBy(moduleIndex, state, subState, cmdState);
			}
			break;

		case ST_COMPLETING:
			if (hasParent_ && escalateComplete_) {
				return pParentLink_->escalateInterruptedBy(moduleIndex, state, subState, cmdState);
			}
			break;

		default:
			break;
	}

	// Flood the hierarchy
	propagateInterruptedBy(moduleIndex, state, subState, cmdState, true);
}

void PackMLModule::propagateInterruptedBy(unsigned long int moduleIndex, PackMLModuleStateEnu state, signed long int subState, PackMLModuleStateEnu cmdState, bool root)
{

	switch (cmdState) { // NOCCM
		case ST_CLEARING:
			if (!(reactToClear_ || overrideClear_ || root)){
				return;
			}
			break;

		case ST_STARTING:
			if (!(reactToStart_ || overrideStart_ || root)){
				return;
			}
			break;

		case ST_STOPPING:
			if (!(reactToStop_ || overrideStop_ || root)){
				return;
			}
			break;

		case ST_ABORTING:
			if (!(reactToAbort_ || overrideAbort_ || root)){
				return;
			}
			break;

		case ST_HOLDING:
			if (!(reactToHold_ || overrideHold_ || root)){
				return;
			}
			break;

		case ST_UNHOLDING:
			if (!(reactToUnhold_ || overrideUnhold_ || root)){
				return;
			}
			break;

		case ST_SUSPENDING:
			if (!(reactToSuspend_ || overrideSuspend_ || root)){
				return;
			}
			break;

		case ST_UNSUSPENDING:
			if (!(reactToUnsuspend_ || overrideUnsuspend_ || root)){
				return;
			}
			break;

		case ST_RESETTING:
			if (!(reactToReset_ || overrideReset_ || root)){
				return;
			}
			break;

		case ST_COMPLETING:
			if (!(reactToComplete_ || overrideComplete_ || root)){
				return;
			}
			break;

		default:
			break;
	}

	interruptedByIndex_ = moduleIndex;
	interruptedInState_ = state;
	interruptedInSubState_ = subState;

	for (unsigned short i = 0; i < childCount_; ++i) {
		childLinks_[i]->propagateInterruptedBy(moduleIndex, state, subState, cmdState, false);
	}

}

void PackMLModule::setInterruptedBy(PackMLModule* pPackMLModule, PackMLModuleStateEnu cmdState)
{
	escalateInterruptedBy(pPackMLModule->getModuleIndex(), pPackMLModule->getCurrentState(), pPackMLModule->getCurrentSubState(), cmdState);
}

		// -----------------------------------------------------------------------------

void PackMLModule::updatePackMLModel_()
{

	switch (stateCurrent_) { // NOCCM
		case ST_UNDEFINED:
			break;

		case ST_STOPPING:
		case ST_CLEARING:
			if (abort_) {
				executeCmd_(ST_ABORTING);
			}
			else if (stateComplete_) {
				executeActingState_(ST_STOPPED);
			}
			else if (needParentSynch(stateCurrent_)) {
				setWaitingFor_(stateCurrent_);
			}
			break;

		case ST_STOPPED:
			checkActivationCondition_();
			if (abort_) {
				executeCmd_(ST_ABORTING);
			}
			else if (stateComplete_) {
				if (reset_) {
					executeCmd_(ST_RESETTING);
				}
				else if (deactivate_) {
					executeCmd_(ST_DEACTIVATING);
				}
			}
			else if (reset_ || deactivate_) {
				if(reset_){
					setWaitingFor_(ST_RESETTING);
				} else {
					setWaitingFor_(ST_DEACTIVATING);
				}
			}
			break;

		case ST_IDLE:
			if (abort_) {
				executeCmd_(ST_ABORTING);
			}
			else if (stateComplete_) {
				if (stop_) {
					executeCmd_(ST_STOPPING);
				}
				else if (start_) {
					executeCmd_(ST_STARTING);
				}
			}
			else if (stop_ || start_) {
				if(stop_){
					setWaitingFor_(ST_STOPPING);
				} else {
					setWaitingFor_(ST_STARTING);
				}
			}
			break;

		case ST_SUSPENDED:
			if (abort_) {
				executeCmd_(ST_ABORTING);
			}
			else if (stateComplete_) {
				if (stop_) {
					executeCmd_(ST_STOPPING);
				}
				else if (complete_) {
					executeCmd_(ST_COMPLETING);
				}
				else if (hold_){
					executeCmd_(ST_HOLDING);
				}
				else if (unsuspend_){
					executeCmd_(ST_UNSUSPENDING);
				}
			}
			else if (stop_ || unsuspend_ || hold_ || complete_) {
				if(stop_){
					setWaitingFor_(ST_STOPPING);
				} else if(unsuspend_){
					setWaitingFor_(ST_UNSUSPENDING);
				} else if(hold_){
					setWaitingFor_(ST_HOLDING);
				} else {
					setWaitingFor_(ST_COMPLETING);
				}
			}
			break;

		case ST_EXECUTE:
			if (abort_) {
				executeCmd_(ST_ABORTING);
			}
			else if (stateComplete_) {
				if (stop_) {
					executeCmd_(ST_STOPPING);
				}
				else if (complete_) {
					executeCmd_(ST_COMPLETING);
				}
				else if (hold_) {
					executeCmd_(ST_HOLDING);
				}
				else if (suspend_) {
					executeCmd_(ST_SUSPENDING);
				}
			}
			else if (stop_ || suspend_ || hold_ || complete_) {
				if(stop_){
					setWaitingFor_(ST_STOPPING);
				} else if(suspend_){
					setWaitingFor_(ST_SUSPENDING);
				} else if(hold_){
					setWaitingFor_(ST_HOLDING);
				} else {
					setWaitingFor_(ST_COMPLETING);
				}
			}
			break;

		case ST_ABORTING:
			if (stateComplete_) {
				executeActingState_(ST_ABORTED);
			}
			else if (needParentSynch(stateCurrent_)) {
				setWaitingFor_(stateCurrent_);
			}
			break;

		case ST_ABORTED:
			checkActivationCondition_();
			if (stateComplete_) {
				if (clear_) {
					executeCmd_(ST_CLEARING);
				}
				else if (deactivate_) {
					executeCmd_(ST_DEACTIVATING);
				}
			}
			else if (clear_ || deactivate_) {
				if(clear_){
					setWaitingFor_(ST_CLEARING);
				} else {
					setWaitingFor_(ST_DEACTIVATING);
				}
			}
			break;

		case ST_HELD:
			if (abort_) {
				executeCmd_(ST_ABORTING);
			}
			else if (stateComplete_) {
				if (stop_) {
					executeCmd_(ST_STOPPING);
				}
				else if (complete_) {
					executeCmd_(ST_COMPLETING);
				}
				else if (unhold_){
					executeCmd_(ST_UNHOLDING);
				}
			}
			else if (stop_ || unhold_ || complete_) {
				if(stop_){
					setWaitingFor_(ST_STOPPING);
				} else if(unhold_){
					setWaitingFor_(ST_UNHOLDING);
				} else {
					setWaitingFor_(ST_COMPLETING);
				}
			}
			break;

		case ST_STARTING:
		case ST_UNHOLDING:
		case ST_UNSUSPENDING:
			if (abort_) {
				executeCmd_(ST_ABORTING);
			}
			else if (stateComplete_) {
				if (stop_) {
					executeCmd_(ST_STOPPING);
				}
				else {
					executeActingState_(ST_EXECUTE);
				}
			}
			else if (needParentSynch(stateCurrent_)) {
				setWaitingFor_(stateCurrent_);
			}
			break;

		case ST_RESETTING:
			if (abort_) {
				executeCmd_(ST_ABORTING);
			}
			else if (stateComplete_) {
				if (stop_) {
					executeCmd_(ST_STOPPING);
				}
				else {
					executeActingState_(ST_IDLE);
				}
			}
			else if (needParentSynch(stateCurrent_)) {
				setWaitingFor_(stateCurrent_);
			}
			break;

		case ST_COMPLETING:
			if (abort_) {
				executeCmd_(ST_ABORTING);
			}
			else if (stateComplete_) {
				if (stop_) {
					executeCmd_(ST_STOPPING);
				}
				else {
					executeActingState_(ST_COMPLETE);
				}
			}
			else if (needParentSynch(stateCurrent_)) {
				setWaitingFor_(stateCurrent_);
			}
			break;

		case ST_HOLDING:
			if (abort_) {
				executeCmd_(ST_ABORTING);
			}
			else if (stateComplete_) {
				if (stop_) {
					executeCmd_(ST_STOPPING);
				}
				else {
					executeActingState_(ST_HELD);
				}
			}
			else if (needParentSynch(stateCurrent_)) {
				setWaitingFor_(stateCurrent_);
			}
			break;

		case ST_SUSPENDING:
			if (abort_) {
				executeCmd_(ST_ABORTING);
			}
			else if (stateComplete_) {
				if (stop_) {
					executeCmd_(ST_STOPPING);
				}
				else {
					executeActingState_(ST_SUSPENDED);
				}
			}
			else if (needParentSynch(stateCurrent_)) {
				setWaitingFor_(stateCurrent_);
			}
			break;

		case ST_COMPLETE:
			if (abort_) {
				executeCmd_(ST_ABORTING);
			}
			else if (stateComplete_) {
				if (stop_) {
					executeCmd_(ST_STOPPING);
				}
				else if (reset_) {
					executeCmd_(ST_RESETTING);
				}
			}
			else if (stop_ || reset_) {
				if(stop_){
					setWaitingFor_(ST_STOPPING);
				} else {
					setWaitingFor_(ST_RESETTING);
				}
			}
			break;

		case ST_DEACTIVATING:
			if (stateComplete_) {
				executeActingState_(ST_DEACTIVATED);
			}
			else {
				setWaitingFor_(stateCurrent_);
			}
			break;

		case ST_DEACTIVATED:
			checkActivationCondition_();
			if (stateComplete_) {
				if (activate_) {
					executeCmd_(ST_ACTIVATING);
				}
			}
			else if (activate_) {
				setWaitingFor_(ST_ACTIVATING);
			}
			break;

		case ST_ACTIVATING:
			if (stateComplete_) {
				executeActingState_(ST_STOPPED);
			}
			else {
				setWaitingFor_(stateCurrent_);
			}
			break;
	}
}

		// -----------------------------------------------------------------------------

void PackMLModule::checkActivationCondition_()
{

	switch (activationCondition_) {
		case 0:
			activate_ = true;
			break;
		case 1: // by parent: do nothing
			break;
		case 2:
			activate_ = activationPv_;;
			deactivate_ = !activate_;
			break;

		default:
			break;
	}

}

		// -----------------------------------------------------------------------------
```

### Program Logical/Program (IEC)

#### Variables.var
```iecst
VAR
	local2 : USINT;
	local1 : USINT;
	counter : USINT;
END_VAR
```

#### Main.st
```iecst
PROGRAM _INIT
	(* Insert code here *)
	local1;
	local2;
	gVar;
END_PROGRAM

PROGRAM _CYCLIC
	(* Insert code here *)
	 counter := counter + 1;
END_PROGRAM

PROGRAM _EXIT
	(* Insert code here *)

END_PROGRAM
```

### RevInfoGlobal.var
```iecst
VAR CONSTANT
	project : STRING[80] := 'DevOpsDemo';
	buildConfiguration : STRING[80] := 'Config1';
	branchName : STRING[80] := 'main';
	tag : STRING[80] := 'v.0.0.4';
	revision : STRING[80] := 'v.0.0.4';
	revisionDate : STRING[80] := '2026-07-08 15:57:29 +0200';
	revisionAuthor : STRING[80] := 'BRGLOBAL\andersenm';
	uncommittedChanges : STRING[80] := '9 files changed, 22 insertions(+), 8 deletions(-)';
	buildDate : STRING[80] := '2026-07-09 11:55:11';
	builder : STRING[80] := 'andersenm';
	commitID : STRING[80] := '63e93e9a43a964874f1086b798fe18c14229c306';
END_VAR
```

### Program Logical/RevInfo/RevInfo (IEC, version 1.0.0)

#### revInfo.st - Init, cyclic, exit code
```iecst
PROGRAM _INIT

	// Instantiation of variables
	// Use variables for e.g. logger, Machine Settings recipe or to a diagnostics HMI page
	project;
	buildConfiguration;
	branchName;
	tag;
	revision;
	revisionDate;
	revisionAuthor;
	uncommittedChanges;
	buildDate;
	builder;
	commitID;

END_PROGRAM

PROGRAM _CYCLIC

END_PROGRAM

PROGRAM _EXIT

END_PROGRAM
```

### Program Logical/EM_Capper/EM_Capper (IEC)

#### local.var
```iecst
VAR
	em : {REDUND_UNREPLICABLE} EquipmentModule;
	Axis : MpAxisBasic;
	Parameters : MpAxisBasicParType;
	simulateAxisError : BOOL;
END_VAR
```

#### alarm.st
```iecst
ACTION alarm:

	IF (*Axis.Error OR*) simulateAxisError THEN // Comment out "real axis error" because it is a test project with no real axis
		em.Command.Abort := TRUE;
	END_IF

END_ACTION
```

#### local.st
```iecst
PROGRAM _INIT

	em.Setup.Name := 'EM_Capper';
	em.Setup.ParentName := 'Main';

	Parameters.Acceleration := 5000;
	Parameters.Deceleration := 5000;

END_PROGRAM

PROGRAM _CYCLIC

	CASE em.ModeID OF
		MODE_PRODUCTION: producing;
		ELSE em.Command.StateComplete := TRUE;
	END_CASE

	alarm;
	modules;

END_PROGRAM

PROGRAM _EXIT

END_PROGRAM
```

#### modules.st
```iecst
ACTION modules:
	// Put all control modules here

	Axis.Enable := TRUE;
	Axis.MpLink := ADR(gAxis_Capper);
	Axis.Parameters := ADR(Parameters);
	Axis();

	em();

END_ACTION
```

#### producing.st
```iecst
ACTION producing:

	CASE em.StateCurrent OF

		STATE_STOPPING:
			em.StateInfo := 'in state stopping';
			em.Command.StateComplete := TRUE;

		STATE_STOPPED:
			em.StateInfo := 'in state stopped';
			em.Command.StateComplete := TRUE;

		STATE_RESETTING:
			em.Command.StateComplete := TRUE;

		STATE_IDLE:
			em.StateInfo := 'in state idle';
			em.Command.Start := TRUE;
			em.Command.StateComplete := TRUE;

		STATE_STARTING:
			em.StateInfo := 'in state starting';
			em.Command.StateComplete := TRUE;

		STATE_EXECUTE:
			em.StateInfo := 'in state execute';

			em.Command.StateComplete := TRUE;

		STATE_ABORTING:
			em.StateInfo := 'in state aborting';
			em.Command.StateComplete := TRUE;

		STATE_ABORTED:
			em.StateInfo := 'in state aborted';
			em.Command.StateComplete := TRUE;

		STATE_CLEARING:
			em.StateInfo := 'in state clearing';
			em.Command.StateComplete := TRUE;

		ELSE
			em.Command.StateComplete := TRUE;

	END_CASE

END_ACTION
```

### global.var
```iecst
VAR
	gCapperInterface : gCapperInterface_typ;
END_VAR
```

### global.typ
```iecst
TYPE
	gCapperInterface_typ : 	STRUCT
		cmd : gConveyorInterface_cmd_typ;
		status : gConveyorInterface_status_typ;
	END_STRUCT;
	gCapperInterface_cmd_typ : 	STRUCT
		startStation : BOOL;
	END_STRUCT;
	gCapperInterface_status_typ : 	STRUCT
		stationDone : BOOL;
		ready : BOOL;
	END_STRUCT;
END_TYPE
```

### Program Logical/EM_Conveyor/EM_Conveyor (IEC)

#### local.st - Init, cyclic, exit code
```iecst
PROGRAM _INIT

	em.Setup.Name := 'EM_Infeed';
	em.Setup.ParentName := 'Main';

	Parameters.Acceleration := 5000;
	Parameters.Deceleration := 5000;

END_PROGRAM

PROGRAM _CYCLIC

	CASE em.ModeID OF
		MODE_PRODUCTION: producing;
		ELSE em.Command.StateComplete := TRUE;
	END_CASE

	alarm;
	modules;
	simulation;

END_PROGRAM

PROGRAM _EXIT

END_PROGRAM
```

#### producing.st
```iecst
ACTION producing:

	CASE em.StateCurrent OF

		STATE_STOPPED:
			em.StateInfo := 'in state stopped';
			em.Command.StateComplete := TRUE;

		STATE_RESETTING:
			CASE em.SubState OF

				0:
					em.StateInfo := 'Wait for Power on';

					Axis.Power := TRUE;

					IF Axis.PowerOn THEN
						em.SubState := 10;
					END_IF

				10:
					em.StateInfo := 'Wait for homing';

					Axis.Home := TRUE;

					IF Axis.IsHomed THEN
						Axis.Home := FALSE;
						em.SubState := 20;
					END_IF

				20:
					em.Command.StateComplete := TRUE;

			END_CASE

		STATE_IDLE:
			em.StateInfo := 'in state idle';
			em.Command.Start := TRUE;
			em.Command.StateComplete := TRUE;

		STATE_STARTING:
			em.StateInfo := 'in state starting';
			em.Command.StateComplete := TRUE;

		STATE_EXECUTE:

			CASE em.SubState OF

				0:
					em.StateInfo := 'Waiting for bottle';
					IF hw.di_bottleReady THEN
						em.SubState := 10;
					END_IF

				10:
					IF gFillerInterface.status.ready AND gCapperInterface.status.ready THEN
						em.SubState := 20;
					END_IF

				20:
					em.StateInfo := 'Start conveyor and wait for bottle to leave photosensor';

					Axis.MoveAdditive := TRUE;
					Parameters.Velocity := 82.0;
					Parameters.Distance := 100.0;

					IF NOT hw.di_bottleReady THEN
						em.SubState := 30;
					END_IF

				30:
					em.StateInfo := 'Wait for axis movement to finish';

					IF Axis.MoveDone THEN
						Axis.MoveAdditive := FALSE;
						em.SubState := 40;
					END_IF

				40:
					em.StateInfo := 'Wait for stations to finish';

					gFillerInterface.cmd.startStation := TRUE;
					gCapperInterface.cmd.startStation := TRUE;

					IF gFillerInterface.status.stationDone AND gCapperInterface.status.stationDone THEN
						gFillerInterface.cmd.startStation := FALSE;
						gCapperInterface.cmd.startStation := FALSE;
						productionCycleCount := productionCycleCount + 1;
						em.SubState := 0;
					END_IF

			END_CASE
			em.Command.StateComplete := TRUE;

		STATE_STOPPING,STATE_ABORTING:
			em.StateInfo := 'in state aborting/stopping';
			Axis.Power := FALSE;
			Axis.Home := FALSE;
			em.Command.StateComplete := TRUE;

		STATE_ABORTED:
			em.StateInfo := 'in state aborted';
			em.Command.StateComplete := TRUE;

		STATE_CLEARING:
			em.StateInfo := 'in state clearing';
			em.Command.StateComplete := TRUE;

		ELSE
			em.Command.StateComplete := TRUE;

	END_CASE

END_ACTION
```

#### alarm.st
```iecst
ACTION alarm:

	IF (*Axis.Error OR *)simulateAxisError THEN // Comment out "real axis error" because it is a test project with no real axis
		em.Command.Abort := TRUE;
	END_IF

END_ACTION
```

#### modules.st
```iecst
ACTION modules:
	// Put all control modules here

	Axis.Enable := TRUE;
	Axis.MpLink := ADR(gAxis_Conveyor);
	Axis.Parameters := ADR(Parameters);
	Axis();

	em();

END_ACTION
```

#### local.typ - Local data types
```iecst
TYPE
	hw_typ : 	STRUCT
		di_bottleReady : BOOL;
	END_STRUCT;
	sim_typ : 	STRUCT
		produce100Bottles : BOOL;
		produce100BottlesWithAxisFault : BOOL;
		axisFaultInjected : BOOL;
		lastCycleCount : UDINT;
	END_STRUCT;
END_TYPE
```

#### local.var - Local variables
```iecst
VAR
	em : {REDUND_UNREPLICABLE} EquipmentModule;
	Axis : MpAxisBasic;
	Parameters : MpAxisBasicParType;
	hw : hw_typ;
	sim : sim_typ;
	productionCycleCount : UDINT;
	simulateAxisError : BOOL;
	TON_simulateBottles : TON;
END_VAR
```

#### simulation.st - not listed in the package file held
```iecst
ACTION simulation:

	IF gIsSimulation THEN

		IF EDGEPOS(sim.produce100Bottles) THEN
			sim.lastCycleCount := productionCycleCount;
		END_IF

		IF sim.produce100Bottles THEN
			IF productionCycleCount >= (sim.lastCycleCount+100) THEN
				sim.produce100Bottles := FALSE;
				hw.di_bottleReady := FALSE;
			ELSIF em.SubState = 0 OR em.SubState = 10 THEN
				hw.di_bottleReady := TRUE;
			ELSE
				hw.di_bottleReady := FALSE;
			END_IF

		END_IF

		IF EDGEPOS(sim.produce100BottlesWithAxisFault) THEN
			sim.lastCycleCount := productionCycleCount;
			sim.axisFaultInjected := FALSE;
		END_IF

		IF sim.produce100BottlesWithAxisFault THEN
			IF productionCycleCount >= (sim.lastCycleCount+100) THEN
				sim.produce100BottlesWithAxisFault := FALSE;
				hw.di_bottleReady := FALSE;
			ELSE
				IF productionCycleCount >= (sim.lastCycleCount+25) AND NOT sim.axisFaultInjected THEN
					simulateAxisError := TRUE;
					sim.axisFaultInjected := TRUE;
				END_IF

				IF em.SubState = 0 OR em.SubState = 10 THEN
					hw.di_bottleReady := TRUE;
				ELSE
					hw.di_bottleReady := FALSE;
				END_IF
			END_IF
		END_IF

	ELSE
		// On real hw just always simulate that a bottle is there. (Only because it is a test machine)
		IF em.StateCurrent = STATE_EXECUTE THEN

			IF em.SubState = 0 OR em.SubState = 10 THEN
				hw.di_bottleReady := TRUE;
			ELSE
				hw.di_bottleReady := FALSE;
			END_IF

		END_IF
	END_IF

END_ACTION
```

### global.var
```iecst
VAR
	gConveyorInterface : gConveyorInterface_typ;
END_VAR
```

### global.typ
```iecst
TYPE
	gConveyorInterface_typ : 	STRUCT
		cmd : gConveyorInterface_cmd_typ;
		status : gConveyorInterface_status_typ;
	END_STRUCT;
	gConveyorInterface_cmd_typ : 	STRUCT
		startStation : BOOL;
	END_STRUCT;
	gConveyorInterface_status_typ : 	STRUCT
		stationDone : BOOL;
		ready : BOOL;
	END_STRUCT;
END_TYPE
```

### Program Logical/EM_Filler/EM_Filler (IEC)

#### local.var
```iecst
VAR
	em : {REDUND_UNREPLICABLE} EquipmentModule;
	hw : hw_typ;
	TON_0 : TON;
END_VAR
```

#### local.st
```iecst
PROGRAM _INIT

	em.Setup.Name := 'EM_Filler';
	em.Setup.ParentName := 'Main';

END_PROGRAM

PROGRAM _CYCLIC

	CASE em.ModeID OF
		MODE_PRODUCTION: producing;
		ELSE em.Command.StateComplete := TRUE;
	END_CASE

	alarm;
	modules;

END_PROGRAM

PROGRAM _EXIT

END_PROGRAM
```

#### producing.st
```iecst
ACTION producing:

	CASE em.StateCurrent OF

		STATE_STOPPED:
			em.StateInfo := 'in state stopped';
			em.Command.StateComplete := TRUE;

		STATE_RESETTING:
			gFillerInterface.status.ready := FALSE;
			em.Command.StateComplete := TRUE;

		STATE_IDLE:
			em.StateInfo := 'in state idle';
			em.Command.Start := TRUE;
			em.Command.StateComplete := TRUE;

		STATE_STARTING:
			em.StateInfo := 'in state starting';
			em.Command.StateComplete := TRUE;

		STATE_EXECUTE:

			CASE em.SubState OF

				0:
					em.StateInfo := 'Ready. Waiting for command';

					IF gFillerInterface.cmd.startStation THEN
						TON_0.IN := FALSE;
						TON_0();
						em.SubState := 10;
					END_IF
					gFillerInterface.status.ready := em.SubState=0;

				10:
					em.StateInfo := 'Filling bottle';

					hw.do_fillBottle := TRUE;

					TON_0.IN := TRUE;
					TON_0.PT := T#250ms;
					TON_0();

					IF TON_0.Q THEN
						hw.do_fillBottle := FALSE;
						gFillerInterface.status.stationDone := TRUE;
						em.SubState := 20;
					END_IF

				20:
					em.StateInfo := 'Wait for command to be false';

					IF NOT gFillerInterface.cmd.startStation THEN
						gFillerInterface.status.stationDone := FALSE;
						em.SubState := 0;
					END_IF

			END_CASE

			em.Command.StateComplete := TRUE;

		STATE_STOPPING,STATE_ABORTING:
			em.StateInfo := 'in state aborting/stopping';
			em.Command.StateComplete := TRUE;

		STATE_ABORTED:
			em.StateInfo := 'in state aborted';
			em.Command.StateComplete := TRUE;

		STATE_CLEARING:
			em.StateInfo := 'in state clearing';
			em.Command.StateComplete := TRUE;

		ELSE
			em.Command.StateComplete := TRUE;

	END_CASE

END_ACTION
```

### global.var
```iecst
VAR
	gFillerInterface : gFillerInterface_typ;
END_VAR
```

### global.typ
```iecst
TYPE
	gFillerInterface_typ : 	STRUCT
		cmd : gFillerInterface_cmd_typ;
		status : gFillerInterface_status_typ;
	END_STRUCT;
	gFillerInterface_cmd_typ : 	STRUCT
		startStation : BOOL;
	END_STRUCT;
	gFillerInterface_status_typ : 	STRUCT
		stationDone : BOOL;
		ready : BOOL;
	END_STRUCT;
END_TYPE
```

### Program Logical/EM_Infeed/EM_Infeed (IEC)

#### local.st
```iecst
PROGRAM _INIT

	em.Setup.Name := 'EM_Infeed';
	em.Setup.ParentName := 'Main';

END_PROGRAM

PROGRAM _CYCLIC

	CASE em.ModeID OF
		MODE_PRODUCTION: producing;
		ELSE em.Command.StateComplete := TRUE;
	END_CASE

	alarm;
	modules;

END_PROGRAM

PROGRAM _EXIT

END_PROGRAM
```

#### modules.st
```iecst
ACTION modules:
	// Put all control modules here

	Axis.Enable := TRUE;
	Axis.MpLink := ADR(gAxis_Infeed);
	Axis.Parameters := ADR(Parameters);
	Axis();

	em();

END_ACTION
```

#### producing.st
```iecst
ACTION producing:

	CASE em.StateCurrent OF

		STATE_STOPPING:
			em.StateInfo := 'in state stopping';
			em.Command.StateComplete := TRUE;

		STATE_STOPPED:
			em.StateInfo := 'in state stopped';
			em.Command.StateComplete := TRUE;

		STATE_RESETTING:
			CASE em.SubState OF

				0:
					Axis.Power := TRUE;

					IF Axis.PowerOn THEN
						em.SubState := 10;
					END_IF

				10:
					em.Command.StateComplete := TRUE;

			END_CASE

		STATE_IDLE:
			em.StateInfo := 'in state idle';
			em.Command.Start := TRUE;
			em.Command.StateComplete := TRUE;

		STATE_STARTING:
			em.StateInfo := 'in state starting';
			em.Command.StateComplete := TRUE;

		STATE_EXECUTE:
			em.StateInfo := 'in state execute';

			CASE em.SubState OF

				0:
					// Example usage.
					Axis.MoveAdditive := TRUE;
					Parameters.Distance := 100.0; // 100mm
					IF Axis.MoveDone THEN
						Axis.MoveAdditive := FALSE;
						em.SubState := 10;
					END_IF

				10:
					// no code yet

			END_CASE
			em.Command.StateComplete := TRUE;

		STATE_ABORTING:
			em.StateInfo := 'in state aborting';
			em.Command.StateComplete := TRUE;

		STATE_ABORTED:
			em.StateInfo := 'in state aborted';
			em.Command.StateComplete := TRUE;

		STATE_CLEARING:
			em.StateInfo := 'in state clearing';
			em.Command.StateComplete := TRUE;

		ELSE
			em.Command.StateComplete := TRUE;

	END_CASE

END_ACTION
```

### Program Logical/EM_Outfeed/EM_Outfeed (IEC)

#### local.st
```iecst
PROGRAM _INIT

	em.Setup.Name := 'EM_Outfeed';
	em.Setup.ParentName := 'Main';

END_PROGRAM

PROGRAM _CYCLIC

	CASE em.ModeID OF
		MODE_PRODUCTION: producing;
		ELSE em.Command.StateComplete := TRUE;
	END_CASE

	alarm;
	modules;

END_PROGRAM

PROGRAM _EXIT

END_PROGRAM
```

### Program Logical/Main/Main (IEC)

#### local.st - Init, cyclic, exit code
```iecst
PROGRAM _INIT

	em.Setup.Name := 'Main';
	gIsSimulation := DiagCpuIsARsim();

END_PROGRAM

PROGRAM _CYCLIC

	CASE em.ModeID OF
		MODE_PRODUCTION: producing;
		ELSE em.Command.StateComplete := TRUE;
	END_CASE

	alarm;
	modules;
	simulation;

END_PROGRAM

PROGRAM _EXIT
	httpStateService.enable := FALSE;
	httpStateService();

END_PROGRAM
```

#### producing.st
```iecst
ACTION producing:

	CASE em.StateCurrent OF

		STATE_STOPPING:
			em.StateInfo := 'in state stopping';
			em.Command.StateComplete := TRUE;

		STATE_STOPPED:
			em.StateInfo := 'in state stopped';

			IF hmi.startMachine THEN
				hmi.startMachine := FALSE;
				em.Command.Reset := TRUE;
			END_IF
			em.Command.StateComplete := TRUE;

		STATE_RESETTING:
			em.Command.StateComplete := TRUE;

		STATE_IDLE:
			em.StateInfo := 'in state idle';
			em.Command.Start := TRUE;
			em.Command.StateComplete := TRUE;

		STATE_STARTING:
			em.StateInfo := 'in state starting';
			em.Command.StateComplete := TRUE;

		STATE_EXECUTE:
			em.StateInfo := 'in state execute';

			IF hmi.stopMachine THEN
				hmi.stopMachine := FALSE;
				em.Command.Stop := TRUE;
			END_IF
			em.Command.StateComplete := TRUE;

		STATE_ABORTING:
			em.StateInfo := 'in state aborting';
			em.Command.StateComplete := TRUE;

		STATE_ABORTED:
			em.StateInfo := 'in state aborted';

			IF hmi.clearMachine THEN
				hmi.clearMachine := FALSE;
				em.Command.Clear := hw.di_EstopOK;
			END_IF
			em.Command.StateComplete := TRUE;

		STATE_CLEARING:
			em.StateInfo := 'in state clearing';
			em.Command.StateComplete := TRUE;

		ELSE
			em.Command.StateComplete := TRUE;

	END_CASE

	IF hmi.abortMachine THEN
		hmi.abortMachine := FALSE;
		em.Command.Abort := TRUE;
	END_IF

END_ACTION
```

#### alarm.st
```iecst
ACTION alarm:

	// No alarms only a demo project
	IF NOT hw.di_EstopOK THEN
		em.Command.Abort := TRUE;
	END_IF

END_ACTION
```

#### modules.st
```iecst
ACTION modules:
	// Put all control modules here

	em();
	machineExecute := (em.StateCurrent = STATE_EXECUTE);

	CASE em.StateCurrent OF
		STATE_UNDEFINED: hmi.packmlState := 'STATE_UNDEFINED';
		STATE_CLEARING: hmi.packmlState := 'STATE_CLEARING';
		STATE_STOPPED: hmi.packmlState := 'STATE_STOPPED';
		STATE_STARTING: hmi.packmlState := 'STATE_STARTING';
		STATE_IDLE: hmi.packmlState := 'STATE_IDLE';
		STATE_SUSPENDED: hmi.packmlState := 'STATE_SUSPENDED';
		STATE_EXECUTE: hmi.packmlState := 'STATE_EXECUTE';
		STATE_STOPPING: hmi.packmlState := 'STATE_STOPPING';
		STATE_ABORTING: hmi.packmlState := 'STATE_ABORTING';
		STATE_ABORTED: hmi.packmlState := 'STATE_ABORTED';
		STATE_HOLDING: hmi.packmlState := 'STATE_HOLDING';
		STATE_HELD: hmi.packmlState := 'STATE_HELD';
		STATE_UNHOLDING: hmi.packmlState := 'STATE_UNHOLDING';
		STATE_SUSPENDING: hmi.packmlState := 'STATE_SUSPENDING';
		STATE_UNSUSPENDING: hmi.packmlState := 'STATE_UNSUSPENDING';
		STATE_RESETTING: hmi.packmlState := 'STATE_RESETTING';
		STATE_COMPLETING: hmi.packmlState := 'STATE_COMPLETING';
		STATE_COMPLETED: hmi.packmlState := 'STATE_COMPLETED';
		STATE_DEACTIVATING: hmi.packmlState := 'STATE_DEACTIVATING';
		STATE_DEACTIVATED: hmi.packmlState := 'STATE_DEACTIVATED';
		STATE_ACTIVATING: hmi.packmlState := 'STATE_ACTIVATING';
	END_CASE

	IF machineExecute THEN
		httpStateResponse := '{"execute":true}';
		httpStateResponseLength := 16;
	ELSE
		httpStateResponse := '{"execute":false}';
		httpStateResponseLength := 17;
	END_IF

	httpStateResponseHeader.protocol := 'HTTP/1.1';
	httpStateResponseHeader.status := '200 OK';
	httpStateResponseHeader.contentType := 'application/json';
	httpStateResponseHeader.contentLength := httpStateResponseLength;
	httpStateResponseHeader.connection := 'Close';
	httpStateResponseHeader.userLine[0].name := 'Access-Control-Allow-Origin';
	httpStateResponseHeader.userLine[0].value := '*';
	httpStateResponseHeader.userLine[1].name := 'Cache-Control';
	httpStateResponseHeader.userLine[1].value := 'no-store';

	httpStateService.enable := TRUE;
	httpStateService.abort := FALSE;
	httpStateService.send := FALSE;
	httpStateService.option := httpOPTION_HTTP_11 OR httpOPTION_SERVICE_TYPE_NAME;
	httpStateService.pServiceName := ADR(httpStateServiceName);
	httpStateService.pResponseHeader := ADR(httpStateResponseHeader);
	httpStateService.pResponseData := ADR(httpStateResponse);
	httpStateService.responseDataLen := httpStateResponseLength;

	IF httpStateService.phase = httpPHASE_RECEIVED THEN
		httpStateService.send := TRUE;
	END_IF

	httpStateService();

	IF Reboot THEN
		Reboot := FALSE;
		SYSreset(1,SYSLIB_WARMSTART);
	END_IF

END_ACTION
```

#### webservice.st
```iecst
ACTION webservice:
	webServiceSend := FALSE;

	IF webServiceEnable AND (hmiHttpService.phase = httpPHASE_RECEIVED) THEN
		IF hmiHttpService.method = httpMETHOD_GET THEN
			IF hmi.conveyorRunning THEN
				webResponseData := '{"running":true}';
			ELSE
				webResponseData := '{"running":false}';
			END_IF;
			webResponseHeader.status := '200 OK';
		ELSE
			webResponseData := '{"running":false}';
			webResponseHeader.status := '405 Method Not Allowed';
			webResponseHeader.userLine[0].name := 'Allow';
			webResponseHeader.userLine[0].value := 'GET';
		END_IF;

		webResponseDataLen := LEN(webResponseData);
		webResponseHeader.protocol := 'HTTP/1.1';
		webResponseHeader.contentType := 'application/json';
		webResponseHeader.contentLength := webResponseDataLen;
		webResponseHeader.connection := 'Close';
		webResponseHeader.userLine[1].name := 'Cache-Control';
		webResponseHeader.userLine[1].value := 'no-store';
		webServiceSend := TRUE;
	END_IF;

	hmiHttpService(
		enable := webServiceEnable,
		send := webServiceSend,
		abort := FALSE,
		option := httpOPTION_HTTP_11 + httpOPTION_SERVICE_TYPE_NAME,
		pServiceName := ADR(webServiceName),
		pUri := 0,
		uriSize := 0,
		pRequestHeader := 0,
		pRequestData := 0,
		requestDataSize := 0,
		pResponseHeader := ADR(webResponseHeader),
		pResponseData := ADR(webResponseData),
		responseDataLen := webResponseDataLen,
		pStatistics := 0,
		pStruct := 0
	);
END_ACTION
```

#### simulation.st
```iecst
ACTION simulation:

END_ACTION
```

#### local.typ - Local data types
```iecst
TYPE
	hmi_typ : 	STRUCT
		startMachine : BOOL;
		stopMachine : BOOL;
		abortMachine : BOOL;
		clearMachine : BOOL;
		packmlState : STRING[40];
	END_STRUCT;
	hw_typ : 	STRUCT
		di_EstopOK : BOOL := TRUE;
	END_STRUCT;
END_TYPE
```

#### local.var - Local variables
```iecst
VAR
	em : {REDUND_UNREPLICABLE} EquipmentModule;
	hmi : hmi_typ;
	hw : hw_typ;
	Reboot : BOOL;
	machineExecute : BOOL; (* TRUE while Main is in STATE_EXECUTE. *)
	httpStateService : httpService; (* AsHttp service that exposes the execute state. *)
	httpStateServiceName : STRING[32] := 'orangeJuiceState.cgi'; (* URI suffix used by the web visu. *)
	httpStateResponse : STRING[32]; (* JSON response body returned to the web visu. *)
	httpStateResponseHeader : httpResponseHeader_t; (* HTTP response header for the JSON state. *)
	httpStateResponseLength : UDINT; (* Response body length [bytes]. *)
END_VAR
```

### Program Logical/Services/Update (IEC)

#### Types.typ
```iecst
TYPE
	hmi_typ : 	STRUCT
		updateReady : BOOL;
		updateSoftware : BOOL;
	END_STRUCT;
END_TYPE
```

#### Variables.var
```iecst
VAR
	DevLink_0 : DevLink;
	state : UINT;
	paramsDevlink : STRING[255];
	deviceUpdateServer : STRING[80];
	ArProjectGetPackageInfo_0 : ArProjectGetPackageInfo;
	ArProjectInstallPackage_0 : ArProjectInstallPackage;
	ArProjectGetInfo_0 : ArProjectGetInfo;
	TON_0 : TON;
	UpdateReady : BOOL;
	UpdateVersion : {REDUND_UNREPLICABLE} STRING[32];
	deviceLocal : STRING[80];
	DirCopy_0 : DirCopy;
	FileCopy_0 : FileCopy;
	FileDelete_0 : FileDelete;
	FileInfo_0 : FileInfo;
	FileCreate_0 : FileCreate;
	FileInfoData_0 : fiFILE_INFO;
	UpdateVersionOnPLC : STRING[32];
	hmi : hmi_typ;
	DirCreate_0 : DirCreate;
END_VAR
```

#### Main.st
```iecst
PROGRAM _INIT

	paramsDevlink := '/SIP=192.168.1.196 /PROTOCOL=ftp /USER=update /PASSWORD=update';
	deviceUpdateServer := 'UPDATE';
	deviceLocal := 'UPDATELOCAL';
	UpdateReady := FALSE;

END_PROGRAM

PROGRAM _CYCLIC

	CASE state OF

		0:
			// Get version on PLC

			ArProjectGetInfo_0.Execute := TRUE;
			ArProjectGetInfo_0();

			IF ArProjectGetInfo_0.Done THEN
				UpdateVersionOnPLC := ArProjectGetInfo_0.ConfigurationVersion;
				ArProjectGetInfo_0.Execute := FALSE;
				ArProjectGetInfo_0();
				state := 5;
			ELSIF ArProjectGetInfo_0.Error THEN
				ArProjectGetInfo_0.Execute := FALSE;
				ArProjectGetInfo_0();
				state := 222;
			END_IF

		5:
			// Create file device to update server

			DevLink_0.enable := TRUE;
			DevLink_0.pDevice := ADR(deviceUpdateServer);
			DevLink_0.pParam := ADR(paramsDevlink);
			DevLink_0();

			IF DevLink_0.status = ERR_OK OR DevLink_0.status = fiERR_DEVICE_ALREADY_EXIST THEN
				DevLink_0.enable := FALSE;
				DevLink_0();
				state := 10;
			ELSIF DevLink_0.status <> ERR_FUB_BUSY THEN
				DevLink_0.enable := FALSE;
				DevLink_0();
				state := 222;
			END_IF

		10:
			TON_0.IN := TRUE;
			TON_0.PT  := T#3s;
			TON_0();

			hmi.updateReady := UpdateReady;

			IF TON_0.Q THEN
				TON_0.IN := FALSE;
				TON_0();
				UpdateReady := FALSE;
				state := 20;
			ELSIF hmi.updateSoftware THEN
				hmi.updateSoftware := FALSE;
				TON_0.IN := FALSE;
				TON_0();

				IF UpdateReady THEN
					state := 50;
				END_IF
			END_IF

		20:
			// Read PIP on update server
			ArProjectGetPackageInfo_0.Execute := TRUE;
			ArProjectGetPackageInfo_0.DeviceName := deviceUpdateServer;
			ArProjectGetPackageInfo_0.FilePath := 'Default_X20CPx68x/pipconfig.xml';
			ArProjectGetPackageInfo_0();

			IF ArProjectGetPackageInfo_0.Done THEN
				ArProjectGetPackageInfo_0.Execute := FALSE;

				UpdateVersion := ArProjectGetPackageInfo_0.ConfigurationVersion;
				// If update on server is different from the version on PLC
				IF ArProjectGetPackageInfo_0.ConfigurationVersion <> UpdateVersionOnPLC THEN
					state := 25;
				ELSE
					state := 10;
				END_IF
				ArProjectGetPackageInfo_0();
			ELSIF ArProjectGetPackageInfo_0.Error THEN
				ArProjectGetPackageInfo_0.Execute := FALSE;
				ArProjectGetPackageInfo_0();
				state := 10;
			END_IF

		25:
			// Read PIP on local server
			ArProjectGetPackageInfo_0.Execute := TRUE;
			ArProjectGetPackageInfo_0.DeviceName := deviceLocal;
			ArProjectGetPackageInfo_0.FilePath := 'Default_X20CPx68x/pipconfig.xml';
			ArProjectGetPackageInfo_0();

			IF ArProjectGetPackageInfo_0.Done OR ArProjectGetPackageInfo_0.Error THEN
				ArProjectGetPackageInfo_0.Execute := FALSE;

				// If PIP on update server is different from the PIP on local server
				IF ArProjectGetPackageInfo_0.ConfigurationVersion <> UpdateVersion THEN
					state := 30;
				ELSE
					// Version already on local server and different from the one on PLC eg. "Ready to update"
					UpdateReady := TRUE;
					state := 10;
				END_IF
				ArProjectGetPackageInfo_0();
			END_IF

		30:
			TON_0.IN := TRUE;
			TON_0.PT  := T#5s;
			TON_0();

			IF TON_0.Q THEN
				TON_0.IN := FALSE;
				TON_0();
				state := 35;
			END_IF

		35:
			// Download update (directory)
			DirCopy_0.enable := TRUE;
			DirCopy_0.pDestDev := ADR(deviceLocal);
			DirCopy_0.pDestDir := ADR('Default_X20CPx68x');
			DirCopy_0.pSrcDev := ADR(deviceUpdateServer);
			DirCopy_0.pSrcDir := ADR('Default_X20CPx68x');
			DirCopy_0.option := fiOVERWRITE;
			DirCopy_0();

			IF DirCopy_0.status = ERR_OK THEN
				DirCopy_0.enable := FALSE;
				DirCopy_0();
				state := 40;
			ELSIF DirCopy_0.status <> ERR_FUB_BUSY THEN
				DirCopy_0.enable := FALSE;
				DirCopy_0();
				state := 10;
			END_IF

		40:
			// Download update (file) arnbcfg.xml
			FileCopy_0.enable := TRUE;
			FileCopy_0.pDestDev := ADR(deviceLocal);
			FileCopy_0.pDest := ADR('arnbcfg.xml');
			FileCopy_0.pSrcDev := ADR(deviceUpdateServer);
			FileCopy_0.pSrc := ADR('arnbcfg.xml');
			FileCopy_0.option := fiOVERWRITE;
			FileCopy_0();

			IF FileCopy_0.status = ERR_OK THEN
				FileCopy_0.enable := FALSE;
				FileCopy_0();
				state := 10;
			ELSIF FileCopy_0.status <> ERR_FUB_BUSY THEN
				FileCopy_0.enable := FALSE;
				FileCopy_0();
				state := 10;
			END_IF

		50:
			// Update
			ArProjectInstallPackage_0.Execute := TRUE;
			ArProjectInstallPackage_0.DeviceName := deviceLocal;
			ArProjectInstallPackage_0.FilePath := 'Default_X20CPx68x/pipconfig.xml';
			ArProjectInstallPackage_0();

			IF ArProjectInstallPackage_0.Done THEN
				ArProjectInstallPackage_0.Execute := FALSE;
				ArProjectInstallPackage_0();
				state := 60;
			ELSIF ArProjectInstallPackage_0.Error THEN
				ArProjectInstallPackage_0.Execute := FALSE;
				ArProjectInstallPackage_0();
				state := 10;
			END_IF

		60:
			// After an update we expect reboot of machine so go here
			TON_0.IN := TRUE;
			TON_0.PT  := T#30s;
			TON_0();

			IF TON_0.Q THEN
				TON_0.IN := FALSE;
				TON_0();
				state := 0;
			END_IF

		222:
			// Unkown error that should be handled
			TON_0.IN := TRUE;
			TON_0.PT  := T#30s;
			TON_0();

			IF TON_0.Q THEN
				TON_0.IN := FALSE;
				TON_0();
				state := 0;
			END_IF

	END_CASE

END_PROGRAM

PROGRAM _EXIT

END_PROGRAM
```

### Program Logical/Services/userfiles (IEC)

#### Variables.var
```iecst
VAR
	DirCopy_0 : DirCopy;
	DirCreate_0 : DirCreate;
	DevLink_0 : DevLink;
	state : USINT;
END_VAR
```

#### Main.st
```iecst
PROGRAM _INIT
	(* Copy files to UserPartition. Only needed due to temp bug in as-cli that don't transfer userfiles correctly *)

END_PROGRAM

PROGRAM _CYCLIC

	CASE state OF

		0:
			// Create "update" directory if it doesnt exist
			DirCreate_0.enable := TRUE;
			DirCreate_0.pDevice := ADR('USER');
			DirCreate_0.pName := ADR('update');
			DirCreate_0();

			IF DirCreate_0.status = ERR_OK OR DirCreate_0.status = fiERR_DIR_ALREADY_EXIST THEN
				DirCreate_0.enable := FALSE;
				DirCreate_0();
				state := 10;
			ELSIF DirCreate_0.status <> ERR_FUB_BUSY THEN
				state := 222;
			END_IF

		10:
			DirCopy_0.enable := TRUE;
			DirCopy_0.pSrcDev := ADR('SYSTEM');
			DirCopy_0.pSrcDir := ADR('ADDONS/DATA/IAT_Data/wwwRoot/BRVisu/Media/web');
			DirCopy_0.pDestDev := ADR('USER');
			DirCopy_0.pDestDir := ADR('web');
			DirCopy_0.option := fiOVERWRITE;
			DirCopy_0();

			IF DirCopy_0.status = ERR_OK THEN
				DirCopy_0.enable := FALSE;
				DirCopy_0();
				state := 20;
			ELSIF DirCopy_0.status <> ERR_FUB_BUSY THEN
				state := 222;
			END_IF

	END_CASE

END_PROGRAM

PROGRAM _EXIT
	(* Insert code here *)

END_PROGRAM
```

### Program Logical/Update

#### Variables.var
```iecst
VAR
	DevLink_0 : DevLink;
	MpBackupCore_0 : MpBackupCore;
	New_Variable : USINT;
	state : UINT;
	paramsDevlink : STRING[255];
END_VAR
```

#### Main.st
```iecst
PROGRAM _INIT

	paramsDevlink := '/SIP=192.168.1.196 /PROTOCOL=ftp /USER=update /PASSWORD=update';

END_PROGRAM

PROGRAM _CYCLIC

	CASE state OF

		0:
			DevLink_0.enable := TRUE;
			DevLink_0.pDevice := ADR('UPDATE');
			DevLink_0.pParam := ADR(paramsDevlink);
			DevLink_0();

			IF DevLink_0.status = ERR_OK THEN
				DevLink_0.enable := FALSE;
				DevLink_0();
				state := 10;
			ELSIF DevLink_0.status <> ERR_FUB_BUSY THEN
				state := 222;
			END_IF

		10:
			MpBackupCore_0.Enable := TRUE;

		222:
			// Unkown error that should be handled

	END_CASE

	MpBackupCore_0.MpLink := ADR(gBackupCore);
	MpBackupCore_0.DeviceName := ADR('UPDATE');
	MpBackupCore_0.Name := ADR(MpBackupCore_0.Info.Automatic.Update.Name);
	MpBackupCore_0();

END_PROGRAM

PROGRAM _EXIT
	(* Insert code here *)

END_PROGRAM
```

Listed in the project but not available here: Logical/Global.typ, Logical/Libraries/BrdkPackML/BrdkPackML.var, Logical/Libraries/PackMLCore/PackMLModuleEnums.hpp, Logical/Libraries/PackMLCore/PackMLModuleSharedInfo.hpp, Logical/Libraries/PackMLCore/PackMLModuleTable.hpp, Logical/Libraries/PackMLCore/AtomicSemaphore.hpp, Logical/RevInfo/RevInfo/types.typ, Logical/RevInfo/RevInfo/variables.var
